FUNCTION_BLOCK BOOL2INT_4 (* Basic Function Block Type *)
  (* Standard: 61499-2 *)
  (* Version 0.0, 7/4/2026, Schneider Electric, Template *)
  PACKAGE SE.Nereda;
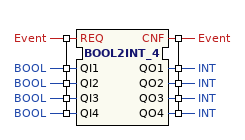
  EVENT_INPUT
    REQ WITH QI1, QI2, QI3, QI4; (* Normal Execution Request *)
  END_EVENT
  EVENT_OUTPUT
    CNF WITH QO1, QO2, QO3, QO4; (* Execution Confirmation *)
  END_EVENT
  VAR_INPUT
    QI1 : BOOL; (* Input event qualifier *)
    QI2 : BOOL;
    QI3 : BOOL;
    QI4 : BOOL;
  END_VAR
  VAR_OUTPUT
    QO1 : INT; (* Output event qualifier *)
    QO2 : INT;
    QO3 : INT;
    QO4 : INT;
  END_VAR
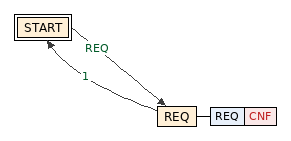
  EC_STATES
    START; (* Initial State *)
    REQ : REQ -> CNF; (* Normal execution *)
  END_STATES
  EC_TRANSITIONS
    START TO REQ := REQ;
    REQ TO START := 1;
  END_TRANSITIONS
  ALGORITHM REQ IN ST: (* Normally executed algorithm *)
;
QO1 := BOOL_TO_INT(QI1);
QO2 := BOOL_TO_INT(QI2);
QO3 := BOOL_TO_INT(QI3);
QO4 := BOOL_TO_INT(QI4);
  END_ALGORITHM
END_FUNCTION_BLOCK
